{attribute 'GeneratedUsingTerminal: ER6002-0002-0021'}
{attribute addProperty BoxType "ER6002-0002-0021"}
{attribute addProperty Id "StatusAT %I*WORD2Data_InAT %I*ARRAY[0..21] OF USINT22"}
{attribute addProperty CRC "3532970676"}
{attribute addProperty Size "24"}
TYPE COM_TxPDO_Map_Inputs_Channel_C252EAC2 EXTENDS InputBase_8311D824 :
STRUCT
	{attribute addProperty Name "Status"}
	Status AT %I* : WORD;
	{attribute addProperty Name "Data_In"}
	Data_In AT %I* : ARRAY[0..21] OF USINT;
END_STRUCT
END_TYPE

(* stored: Version 1.2.0.0, ProductVersion 3.1.4024.9
   DUT COM_TxPDO_Map_Inputs_Channel_C252EAC2: Id {8139e84b-3e8a-4f4a-b2c6-7dadfadc24ab} *)
